//==================================================================================================
//								RJM Maszyny sp. z o.o.
//									13.05.2022
//
//	Obsługa czujnika
//	v1.0	|| TC v 3.1.4024.22		|| - pierwsza wersja
//==================================================================================================
FUNCTION_BLOCK FB_Czujnik_NO IMPLEMENTS I_Czujnik
VAR
	Wejscie 						AT %I* 	: BOOL;
END_VAR

//==================================================================================================
//								RJM Maszyny sp. z o.o.
//									13.05.2022
//
//	Sprawdzenie czy aktywny
//	v1.0	|| TC v 3.1.4024.22		|| - pierwsza wersja
//==================================================================================================
PROPERTY CzyAktywny : BOOL
GET
CzyAktywny 									:= Wejscie;
END_GET
END_PROPERTY

END_FUNCTION_BLOCK

(* stored: Version 1.1.0.1, ProductVersion 3.1.4024.11
   POU FB_Czujnik_NO: Id {fe7f936a-5c93-4035-995a-e10f28bd6ad6}, SpecialFunc None
   Property CzyAktywny: Id {52dbf970-d522-4bcf-b92a-05d4c8a39dcb}
   Get Get: Id {b4293b22-5339-4397-9c81-45b1aba2db51} *)
